{attribute 'GeneratedUsingTerminal: KL2184'}
{attribute addProperty BoxType "KL2184"}
{attribute addProperty Id "Channel_1AT %Q*Channel_460B8C400Channel_2AT %Q*Channel_460B8C400Channel_3AT %Q*Channel_460B8C400Channel_4AT %Q*Channel_460B8C400"}
{attribute addProperty CRC "3835617775"}
{attribute addProperty Size "0"}
TYPE KL2184_E49EE1EF :
STRUCT
	{attribute addProperty Name "Channel_1"}
	Channel_1 : Channel_460B8C40;
	{attribute addProperty Name "Channel_2"}
	Channel_2 : Channel_460B8C40;
	{attribute addProperty Name "Channel_3"}
	Channel_3 : Channel_460B8C40;
	{attribute addProperty Name "Channel_4"}
	Channel_4 : Channel_460B8C40;
END_STRUCT
END_TYPE

(* stored: Version 1.2.0.0, ProductVersion 3.1.4024.9
   DUT KL2184_E49EE1EF: Id {9c58fb74-7ac7-4673-b440-f6ee6ebacefd} *)
